{attribute 'qualified_only'}
{attribute 'strict'}
TYPE eErrorMessage :
(
	eNoError							:= 0,
	eReceivedMessageWithError			:= 1,
	eReceivedMessageIncompatibility		:= 2,
	eCreatedMessageWithError			:= 3
);
END_TYPE

(* stored: Version 1.1.0.1, ProductVersion 3.1.4024.6
   DUT eErrorMessage: Id {4a334745-54f3-401b-a478-9a2515141d66} *)
